fb_ST1K2_PPS_VGC_1(
                         i_stUSG := fb_SP1K2_PAX_PIP_1.q_IG,
                         i_stDSG := fb_ST1K2_PPS_PIP_1.q_IG,
                         i_xDis_DPIlk := FALSE,
                         i_xEPS_OK := TRUE,
                         i_xPMPS_OK := TRUE,
                         i_xExt_OK := TRUE,
                         i_xOverrideMode := xSystemOverrideMode1,
                         io_fbFFHWO := g_FastFaultOutput1, fbArbiter := fbArbiter1);

fb_MR2K2_FLAT_VGC_1(
                         i_stUSG := fb_ST1K2_PPS_PIP_1.q_IG,
                         i_stDSG := fb_MR2K2_FLAT_PIP_1.q_IG,
                         i_xDis_DPIlk := FALSE,
                         i_xEPS_OK := TRUE,
                         i_xPMPS_OK := TRUE,
                         i_xExt_OK := TRUE,
                         i_xOverrideMode := xSystemOverrideMode2,
                         io_fbFFHWO := g_FastFaultOutput2, fbArbiter := fbArbiter2);

fb_MR2K2_FLAT_VGC_2(
                         i_stUSG := fb_MR2K2_FLAT_PIP_1.q_IG,
                         i_stDSG := fb_IM2K2_PPM_PIP_1.q_IG,
                         i_xDis_DPIlk := FALSE,
                         i_xEPS_OK := TRUE,
                         i_xPMPS_OK := TRUE,
                         i_xExt_OK := TRUE,
                         i_xOverrideMode := xSystemOverrideMode2,
                         io_fbFFHWO := g_FastFaultOutput2, fbArbiter := fbArbiter2);

fb_MR3K2_KBH_VGC_1(
                         i_stUSG := fb_IM2K2_PPM_PIP_1.q_IG,
                         i_stDSG := fb_MR3K2_KBH_PIP_1.q_IG,
                         i_xDis_DPIlk := FALSE,
                         i_xEPS_OK := TRUE,
                         i_xPMPS_OK := TRUE,
                         i_xExt_OK := TRUE,
                         i_xOverrideMode := xSystemOverrideMode2,
                         io_fbFFHWO := g_FastFaultOutput2, fbArbiter := fbArbiter2);

fb_MR3K2_KBH_VGC_2(
                         i_stUSG := fb_MR3K2_KBH_PIP_1.q_IG,
                         i_stDSG := fb_IM3K2_PPM_PIP_1.q_IG,
                         i_xDis_DPIlk := FALSE,
                         i_xEPS_OK := TRUE,
                         i_xPMPS_OK := TRUE,
                         i_xExt_OK := TRUE,
                         i_xOverrideMode := xSystemOverrideMode2,
                         io_fbFFHWO := g_FastFaultOutput2, fbArbiter := fbArbiter2);

fb_MR4K2_KBV_VGC_1(
                         i_stUSG := fb_IM3K2_PPM_PIP_1.q_IG,
                         i_stDSG := fb_MR4K2_KBV_PIP_1.q_IG,
                         i_xDis_DPIlk := FALSE,
                         i_xEPS_OK := TRUE,
                         i_xPMPS_OK := TRUE,
                         i_xExt_OK := TRUE,
                         i_xOverrideMode := xSystemOverrideMode2,
                         io_fbFFHWO := g_FastFaultOutput2, fbArbiter := fbArbiter2);

fb_MR4K2_KBV_VGC_2(
                         i_sDevName:='MR4K2_KBV_VGC_2',
                         i_stUSG := fb_MR4K2_KBV_PIP_1.q_IG,
                         i_stDSG := fb_IM5K2_PPM_GCC_1.IG,
                         i_xDis_DPIlk := FALSE,
                         i_xEPS_OK := TRUE,
                         i_xPMPS_OK := TRUE,
                         i_xExt_OK := TRUE,
                         i_xOverrideMode := xSystemOverrideMode2,
                         io_fbFFHWO := g_FastFaultOutput2, fbArbiter := fbArbiter2);

fb_LI3K2_K2B_VWC_1(
                         i_stUSG := fb_TM2K2_K2B_GCC_1.IG,
                         i_stDSG := fb_TM2K2_K2B_GCC_1.IG,
                         i_xDis_DPIlk := FALSE,
                         i_xIsAperture := TRUE,
                         i_xEPS_OK := TRUE,
                         i_xPMPS_OK := TRUE,
                         i_xExt_OK := TRUE,
                         i_xOverrideMode := xSystemOverrideMode2,
                         io_fbFFHWO := g_FastFaultOutput2, fbArbiter := fbArbiter2);

fb_SP1K2_PAX_VGC_1(
                         i_stUSG := fb_SL1K2_EXIT_PIP_1.q_IG,
                         i_stDSG := fb_SP1K2_PAX_PIP_1.q_IG,
                         i_xDis_DPIlk := FALSE,
                         i_xEPS_OK := TRUE,
                         i_xPMPS_OK := TRUE,
                         i_xExt_OK := TRUE,
                         i_xOverrideMode := xSystemOverrideMode1,
                         io_fbFFHWO := g_FastFaultOutput1, fbArbiter := fbArbiter1);

fb_LI2K2_K2A_VWC_1(
                         i_stUSG := fb_IM5K2_PPM_GCC_1.IG,
                         i_stDSG := fb_IM5K2_PPM_GCC_1.IG,
                         i_xDis_DPIlk := FALSE,
                         i_xIsAperture := TRUE,
                         i_xEPS_OK := TRUE,
                         i_xPMPS_OK := TRUE,
                         i_xExt_OK := TRUE,
                         i_xOverrideMode := xSystemOverrideMode2,
                         io_fbFFHWO := g_FastFaultOutput2, fbArbiter := fbArbiter2);

//PAX VRCs
bSP1K2_PAX_VRC_1_ILK := F_TurboGateValve_Protection_ILK(i_Turbo:=fb_SP1K2_PAX_PTM_01.iq_stPtm,
                                               i_stISG:=fb_SP1K2_PAX_GPI_1.PG,
                                               i_stBSG:=RIXS_ROUGH_GPI_01.PG,
                                                 ScrollPump:=RIXS_PRO_01.stPump);
fb_SP1K2_PAX_VRC_1(i_xExtILK_OK:=bSP1K2_PAX_VRC_1_ILK,
            i_xOverrideMode:=xSystemOverrideMode1,
            iq_stValve =>);

bSP1K2_PAX_VRC_2_ILK := F_TurboGateValve_Protection_ILK(i_Turbo:=fb_SP1K2_PAX_PTM_02.iq_stPtm,
                                               i_stISG:=fb_SP1K2_PAX_GPI_2.PG,
                                               i_stBSG:=RIXS_ROUGH_GPI_01.PG,
                                                 ScrollPump:=RIXS_PRO_01.stPump);
fb_SP1K2_PAX_VRC_2(i_xExtILK_OK:=bSP1K2_PAX_VRC_2_ILK,
            i_xOverrideMode:=xSystemOverrideMode1,
            iq_stValve =>);

//Manual Valve, only readback
fb_SP1K2_PAX_VRM_3(i_xExtILK_OK:=TRUE,
            i_xOverrideMode:=xSystemOverrideMode1,
            iq_stValve =>);

// backing PAX chamber
fb_SP1K2_PAX_VRC_4(i_xExtILK_OK :=  qRIXS_PRO_01.st_pro.eState = E_PumpState.pumpRUNNING, i_xOverrideMode := xSystemOverrideMode1, iq_stValve =>)	;


//PAX Turbo Pumps (PTM) ILK
fb_SP1K2_PAX_PTM_01(i_xExtIlkOK:= fb_SP1K2_PAX_VRC_4.M_IsOpen()
                AND F_TurboExtILKLogic_2(Turbo:=fb_SP1K2_PAX_PTM_01.iq_stPTM,BackingGauge:=RIXS_ROUGH_GPI_01.PG, InletGauge:=fb_SP1K2_PAX_GPI_1.PG, ScrollPump:= RIXS_PRO_01.stPump) );

fb_SP1K2_PAX_PTM_02(i_xExtIlkOK:= fb_SP1K2_PAX_VRC_4.M_IsOpen()
                AND F_TurboExtILKLogic_2(Turbo:=fb_SP1K2_PAX_PTM_02.iq_stPTM,BackingGauge:=RIXS_ROUGH_GPI_01.PG, InletGauge:=fb_SP1K2_PAX_GPI_2.PG, ScrollPump:= RIXS_PRO_01.stPump) );


(*********SERIAL COMMUNICATION**********)
(*Pfeiffer pumps*)
//SP1K2_PAX_PTM_01
(*Assign adresses to the pfeiffer controllers connected to this serial terminal*)
stPfeiffer_CTRL_SP1K2_PAX_PTM_01[1].iSerialAddress:= 1;
stPfeiffer_CTRL_SP1K2_PAX_PTM_01[1].xEnableComm:= TRUE;
(*Instanitate the Function block for serial communication with Pfeiffer*)
fbPfeifferCom_SP1K2_PAX_PTM_01(astPfeifferControl:= stPfeiffer_CTRL_SP1K2_PAX_PTM_01,
                              astPfeifferStatus:= stPfeiffer_RBK_SP1K2_PAX_PTM_01,
                              SerialRXBuffer:= SerialRXBuffer_SP1K2_PAX_PTM_01,
                              SerialTXBuffer:= SerialTXBuffer_SP1K2_PAX_PTM_01);
(*Copy Status Pv's into the PTM structure*)
fb_SP1K2_PAX_PTM_01.M_Serial_IO(st_Pfeiffer_RBK:= stPfeiffer_RBK_SP1K2_PAX_PTM_01[1],
                            st_Pfeiffer_CTRL:= stPfeiffer_CTRL_SP1K2_PAX_PTM_01[1]);

//SP1K2_PAX_PTM_02
(*Assign adresses to the pfeiffer controllers connected to this serial terminal*)
stPfeiffer_CTRL_SP1K2_PAX_PTM_02[1].iSerialAddress:= 1;
stPfeiffer_CTRL_SP1K2_PAX_PTM_02[1].xEnableComm:= TRUE;
(*Instanitate the Function block for serial communication with Pfeiffer*)
fbPfeifferCom_SP1K2_PAX_PTM_02(astPfeifferControl:= stPfeiffer_CTRL_SP1K2_PAX_PTM_02,
                              astPfeifferStatus:= stPfeiffer_RBK_SP1K2_PAX_PTM_02,
                              SerialRXBuffer:= SerialRXBuffer_SP1K2_PAX_PTM_02,
                              SerialTXBuffer:= SerialTXBuffer_SP1K2_PAX_PTM_02);
(*Copy Status Pv's into the PTM structure*)
fb_SP1K2_PAX_PTM_02.M_Serial_IO(st_Pfeiffer_RBK:= stPfeiffer_RBK_SP1K2_PAX_PTM_02[1],
                            st_Pfeiffer_CTRL:= stPfeiffer_CTRL_SP1K2_PAX_PTM_02[1]);

// PIP_Gamma Pumps

fb_PC1K1_ZOS_PIP_1(i_stGauge := fb_PC1K1_ZOS_GPI_1.PG, i_xOverrideMode := xSystemOverrideMode1);
fb_MR1K2_SWITCH_PIP_1(i_stGauge := fb_MR1K2_SWITCH_GPI_1.PG, i_xOverrideMode := xSystemOverrideMode1);
fb_TV1K1_PLEG_PIP_1(i_stGauge := fb_TV1K1_PLEG_GPI_1.PG, i_xOverrideMode := xSystemOverrideMode1);
fb_SL1K2_EXIT_PIP_1(i_stGauge := fb_SL1K2_EXIT_GPI_1.PG, i_xOverrideMode := xSystemOverrideMode1);
fb_ST1K2_PPS_PIP_1(i_stGauge := fb_ST1K2_PPS_GPI_1.PG, i_xOverrideMode := xSystemOverrideMode1);
fb_MR2K2_FLAT_PIP_1(i_stGauge := fb_MR2K2_FLAT_GPI_1.PG, i_xOverrideMode := xSystemOverrideMode2);
fb_MR3K2_KBH_PIP_1(i_stGauge := fb_MR3K2_KBH_GPI_1.PG, i_xOverrideMode := xSystemOverrideMode2);
fb_MR4K2_KBV_PIP_1(i_stGauge := fb_MR4K2_KBV_GPI_1.PG, i_xOverrideMode := xSystemOverrideMode2);
fb_TV4K2_PIP_1(i_stGauge := bm_dummy_gauge, i_xOverrideMode := xSystemOverrideMode2);
fb_IM5K2_PPM_PIP_1(i_stGauge := bm_dummy_gauge, i_xOverrideMode := xSystemOverrideMode2);
fb_PA1K2_PIP_1(i_stGauge := bm_dummy_gauge, i_xOverrideMode := xSystemOverrideMode2);
fb_SP1K2_PAX_PIP_1(i_stGauge := fb_ST1K2_PPS_GPI_1.PG, i_xOverrideMode := xSystemOverrideMode1);  //change interlock to SP1K2 GPI once connected

//SIP Pumps
fb_IM2K2_PPM_PIP_1(i_stGauge := bm_dummy_gauge, i_xOverrideMode := xSystemOverrideMode2);
fb_IM3K2_PPM_PIP_1(i_stGauge := bm_dummy_gauge, i_xOverrideMode := xSystemOverrideMode2);
fb_IM4K2_PPM_PIP_1(i_stGauge := bm_dummy_gauge, i_xOverrideMode := xSystemOverrideMode2);
fb_LI2K2_K2A_PIP_1(i_stGauge := bm_dummy_gauge, i_xOverrideMode := xSystemOverrideMode2);
fb_ST3K2_TERM_PIP_1(i_stGauge := bm_dummy_gauge, i_xOverrideMode := xSystemOverrideMode2);

//Fast shutter Valve Interface
vfs_dummy_gauge.xPRESS_OK := TRUE;
vfs_dummy_gauge.rPRESS := 0.0000001;
fb_TV1K2_VFS_Interface(IG:=fb_TV4K2_GFS_1.IG, iq_stValve=> , Veto_Valve:=fb_MR4K2_KBV_VGC_2.iq_stValve, i_xVAC_FAULT_OK=> );
//TV1K2_VFS_Interface(IG:= fb_TV4K2_GFS_1.IG);


//Interface for KFE VAC SP1K1-ZOS-VGC-2
// Update interlock signals for RIX
fb_RIX_ILK(
    VG	:=	fb_PC1K1_ZOS_PIP_1.q_IG, //fb_PC1K1_ZOS_GCC_1.IG,
    ILK	:=	st_RIX_ILK
);

END_PROGRAM

// ---- POUs/FB_PRO_ADS.TcPOU
(* This function block is created for interface devices between different PLC*)
(* Not all the Variables in the original structure is required, just few signals *)
(* The variable values are read via ADS using the symbol name*)
FUNCTION_BLOCK FB_PRO_ADS Extends FB_ADS
VAR_INPUT
    sNetId : String; //NetID of the Destination PLC controller
    nPort : uint; // port number
    sVarName : string;// the variable name of the declared gauge function block.
    iWatchdog:UDINT;//The watchdog variable name written to by the remote plc
END_VAR
VAR_OUTPUT
    {attribute 'pytmc' := 'pv:'}
    st_pro : ST_EbaraDryPump;
    bError: BOOL;
END_VAR
VAR
    fb_CheckWatchdog: FB_CheckWatchdog;
    fb_Read_PRO: FB_ReadAdsSymByName;
    ftReset: F_TRIG;
    xFirstPass: BOOL:= true;
END_VAR

ftReset(CLK:= fb_Read_PRO.bBusy OR xFirstPass);
xFirstPass := false;
(*calling ADS read function*)

//IG.xPRESS_OK := false;

fb_Read_PRO(
    bRead:=ftReset.Q ,
    sNetId:= sNetId,
    nPort:= nPort,
    sVarName:= CONCAT(sVarName,'.stPump'),
    nDestAddr:= ADR(st_pro),
    nLen:= SIZEOF(ST_EbaraDryPump),
    tTimeout:= ,
    eComMode:=eAdsComModeFastCom ,
    bBusy=> ,
    bError=> ,
    nErrorId=> );


(*Error*)
fb_CheckWatchdog(
    bEnable:= TRUE,
    tWatchdogTime:= T#900ms,
    nCnt:= iWatchdog ,
    bWatchdog=> ,
    nLastCnt=> );

bError:= fb_Read_PRO.bError OR fb_CheckWatchdog.bWatchdog;
tErrorPresent(CLK:=bError);

IF (fb_Read_PRO.bError OR fb_CheckWatchdog.bWatchdog) THEN
st_pro.i_xAlarm:= TRUE;
END_IF;

END_FUNCTION_BLOCK

// ---- POUs/PRG_RIX_INTF.TcPOU
PROGRAM PRG_RIX_INTF
VAR
{attribute 'pytmc' := '
        pv: PLC:KFE:RIX:FIM:COMBO:ILK
        io: i;
'}
FB_FIM_ILK	AT%Q*	:	BOOL;
END_VAR

ads_watch_dog(
    sNetId := '172.21.140.47.1.1', // AMS NET ID of the PLC reading from this PLC
    nPort := 851, // ADS port of the PLC reading from this PLC
    sVarName := 'PRG_ADS_Interfaces.i_iWatchdog', // Full name of the UDINT provided to the 'iWatchdog' parameter in the interface functions on the PLC reading from this PLC
);

ads_watch_dog_qrix(
    sNetId := '172.21.140.43.1.1', // AMS NET ID of the PLC reading from this PLC
    nPort := 851, // ADS port of the PLC reading from this PLC
    sVarName := 'PRG_SampleChamber.iWatchdog', // Full name of the UDINT provided to the 'iWatchdog' parameter in the interface functions on the PLC reading from this PLC
);

FB_MR3K2_FIM_ILK(
    VG := fb_MR3K2_KBH_PIP_1.q_IG,
    ILK := ST_MR3K2_FIM_ILK,
);

FB_MR4K2_FIM_ILK(
    VG := fb_MR4K2_KBV_PIP_1.q_IG,
    ILK := ST_MR4K2_FIM_ILK,
);

FB_FIM_ILK := ( ST_MR3K2_FIM_ILK.q_xILK_OK_DO AND ST_MR4K2_FIM_ILK.q_xILK_OK_DO );

END_PROGRAM

// ---- POUs/PRG_Roughing.TcPOU
PROGRAM PRG_Roughing
VAR
END_VAR

// Roughing devices
//MKS 275 Gauges
RIXS_ROUGH_GPI_01.M_SetBits(30518);
RIXS_ROUGH_GPI_01();			// Roughing guage near pro


RIXS_PRO_01(i_stBPGauge := RIXS_ROUGH_GPI_01.PG, i_xVlvOpn := TRUE, i_xExtIlkOK := TRUE);


if( RIXS_PRO_01.stPump.eState = pumpSTARTING ) OR ( RIXS_PRO_01.stPump.eState = pumpRUNNING )
 THEN RIXS_ROUGH_VRO_01.M_Open(TRUE); 
END_IF
RIXS_ROUGH_VRO_01(i_xExtILK_OK:= (RIXS_PRO_01.stPump.eState = pumpRUNNING  OR  RIXS_PRO_01.stPump.eState = pumpSTARTING ), i_xOverrideMode:= , iq_stValve=> );

END_PROGRAM

// ---- POUs/PRG_COM.TcPOU
PROGRAM PRG_COM
VAR

END_VAR

(*Instanitate Serial port com function *)
fbSerialLineControl_SP1K2_PAX_PTM_01(
    Mode:= SERIALLINEMODE_EL6_22B,
    pComIn:= ADR(stComIn_SP1K2_PAX_PTM_01),
    pComOut:= ADR(stComOut_SP1K2_PAX_PTM_01),
    SizeComIn:= UINT_TO_INT(SIZEOF(stComIn_SP1K2_PAX_PTM_01)),
    TxBuffer:= SerialTXBuffer_SP1K2_PAX_PTM_01,
    RxBuffer:= SerialRXBuffer_SP1K2_PAX_PTM_01,
    Error=> ,
    ErrorID=> );

fbSerialLineControl_SP1K2_PAX_PTM_02(
    Mode:= SERIALLINEMODE_EL6_22B,
    pComIn:= ADR(stComIn_SP1K2_PAX_PTM_02),
    pComOut:= ADR(stComOut_SP1K2_PAX_PTM_02),
    SizeComIn:= UINT_TO_INT(SIZEOF(stComIn_SP1K2_PAX_PTM_02)),
    TxBuffer:= SerialTXBuffer_SP1K2_PAX_PTM_02,
    RxBuffer:= SerialRXBuffer_SP1K2_PAX_PTM_02,
    Error=> ,
    ErrorID=> );

END_PROGRAM

// ---- POUs/FB_EXT_ILK.TcPOU
FUNCTION_BLOCK FB_EXT_ILK
VAR_INPUT
    VG	:	ST_VG;
END_VAR
VAR_IN_OUT
    ILK	:	ST_EXT_ILK;
END_VAR
VAR_OUTPUT
END_VAR
VAR
    q_xILK_OK_DO	 AT%Q*	:	BOOL; // Send the signal to indicate that the interlock pressure has been met.
END_VAR

// Indicate that the interlock condition is met.
ILK.xIlkOK 			:= (VG.rPRESS < ILK.rPRO_SP) AND (VG.xPRESS_OK);
// Raise the output signal if the interlock condition is met AND the signal is enabled.
q_xILK_OK_DO		:= (VG.rPRESS < ILK.rPRO_SP) AND (VG.xPRESS_OK) AND (ILK.xIlk_sw);
// Se PV  indicating the output status
ILK.q_xILK_OK_DO	:= q_xILK_OK_DO;

END_FUNCTION_BLOCK

// ---- CheckBounds.TcPOU
// Implicitly generated code : DO NOT EDIT
FUNCTION CheckBounds : DINT
VAR_INPUT
    index, lower, upper: DINT;
END_VAR

// Implicitly generated code : Only an Implementation suggestion
{noflow}
IF  index < lower THEN
    CheckBounds := lower;
ELSIF  index > upper THEN
    CheckBounds := upper;
ELSE
    CheckBounds := index;
END_IF
{flow}

END_FUNCTION

// ---- CheckDivDInt.TcPOU
// Implicitly generated code : DO NOT EDIT
FUNCTION CheckDivDInt : DINT
VAR_INPUT
    divisor:DINT;
END_VAR

// Implicitly generated code : Only an Implementation suggestion
{noflow}
IF divisor = 0 THEN
    CheckDivDInt:=1;
ELSE
    CheckDivDInt:=divisor;
END_IF;
{flow}

END_FUNCTION

// ---- CheckDivLInt.TcPOU
// Implicitly generated code : DO NOT EDIT
FUNCTION CheckDivLInt : LINT
VAR_INPUT
    divisor:LINT;
END_VAR

// Implicitly generated code : Only an Implementation suggestion
{noflow}
IF divisor = 0 THEN
    CheckDivLInt:=1;
ELSE
    CheckDivLInt:=divisor;
END_IF;
{flow}

END_FUNCTION

// ---- CheckDivLReal.TcPOU
// Implicitly generated code : DO NOT EDIT
FUNCTION CheckDivLReal : LREAL
VAR_INPUT
    divisor:LREAL;
END_VAR

// Implicitly generated code : Only an Implementation suggestion
{noflow}
IF divisor = 0 THEN
    CheckDivLReal:=1;
ELSE
    CheckDivLReal:=divisor;
END_IF;
{flow}

END_FUNCTION

// ---- CheckDivReal.TcPOU
// Implicitly generated code : DO NOT EDIT
FUNCTION CheckDivReal : REAL
VAR_INPUT
    divisor:REAL;
END_VAR

// Implicitly generated code : Only an Implementation suggestion
{noflow}
IF divisor = 0 THEN
    CheckDivReal:=1;
ELSE
    CheckDivReal:=divisor;
END_IF;
{flow}

END_FUNCTION

// ---- CheckLRangeSigned.TcPOU
// Implicitly generated code : DO NOT EDIT
FUNCTION CheckLRangeSigned : LINT
VAR_INPUT
    value, lower, upper: LINT;
END_VAR

// Implicitly generated code : Only an Implementation suggestion
{noflow}
IF (value < lower) THEN
    CheckLRangeSigned := lower;
ELSIF(value > upper) THEN
    CheckLRangeSigned := upper;
ELSE
    CheckLRangeSigned := value;
END_IF

{flow}

END_FUNCTION

// ---- CheckLRangeUnsigned.TcPOU
// Implicitly generated code : DO NOT EDIT
FUNCTION CheckLRangeUnsigned : ULINT
VAR_INPUT
    value, lower, upper: ULINT;
END_VAR

// Implicitly generated code : Only an Implementation suggestion
{noflow}
IF (value < lower) THEN
    CheckLRangeUnsigned := lower;
ELSIF(value > upper) THEN
    CheckLRangeUnsigned := upper;
ELSE
    CheckLRangeUnsigned := value;
END_IF
{flow}

END_FUNCTION

// ---- CheckPointer.TcPOU
// Implicitly generated code : DO NOT EDIT
FUNCTION CheckPointer : POINTER TO BYTE
VAR_INPUT
    ptToTest : POINTER TO BYTE; // Destination address of the pointer
    iSize : DINT;		        // Size of the type the pointer points to. (e.g: 20 for POINTER TO ARRAY [0..9] OF INT)
    iGran : DINT;		        // Granularity of the pointer access. This is the size of the biggest non-structured data type in the type the pointer points to. (e.g: 2 for POINTER TO ARRAY [0..9] OF INT)
    bWrite: BOOL;		        // Indicates read or write Access. TRUE = write access.
END_VAR

// Implicitly generated code : Only an Implementation suggestion
{noflow}
IF ptToTest=0 THEN
    ADSLOGSTR(ADSLOG_MSGTYPE_ERROR OR ADSLOG_MSGTYPE_STRING,'CheckPointer failed due to invalid address.','');
ELSIF iSize<=0 THEN
    ADSLOGSTR(ADSLOG_MSGTYPE_ERROR OR ADSLOG_MSGTYPE_STRING,'CheckPointer failed due to invalid size.','');
ELSIF iGran<=0 THEN
    ADSLOGSTR(ADSLOG_MSGTYPE_ERROR OR ADSLOG_MSGTYPE_STRING,'CheckPointer failed due to invalid granularity.','');
// -> Please note that the following memory area check is time consuming:
//ELSIF F_CheckMemoryArea(pData:=ptToTest,nSize:=DINT_TO_UDINT(iSize)) = E_TcMemoryArea.Unknown THEN
//    ADSLOGSTR(ADSLOG_MSGTYPE_ERROR OR ADSLOG_MSGTYPE_STRING,'CheckPointer failed due to unknown memory area.','');
END_IF
CheckPointer := ptToTest;
{flow}

END_FUNCTION

// ---- CheckRangeSigned.TcPOU
// Implicitly generated code : DO NOT EDIT
FUNCTION CheckRangeSigned : DINT
VAR_INPUT
    value, lower, upper: DINT;
END_VAR

// Implicitly generated code : Only an Implementation suggestion
{noflow}
IF (value < lower) THEN
    CheckRangeSigned := lower;
ELSIF(value > upper) THEN
    CheckRangeSigned := upper;
ELSE
    CheckRangeSigned := value;
END_IF
{flow}

END_FUNCTION

// ---- CheckRangeUnsigned.TcPOU
// Implicitly generated code : DO NOT EDIT
FUNCTION CheckRangeUnsigned : UDINT
VAR_INPUT
    value, lower, upper: UDINT;
END_VAR

// Implicitly generated code : Only an Implementation suggestion
{noflow}
IF (value < lower) THEN
    CheckRangeUnsigned := lower;
ELSIF(value > upper) THEN
    CheckRangeUnsigned := upper;
ELSE
    CheckRangeUnsigned := value;
END_IF
{flow}

END_FUNCTION
